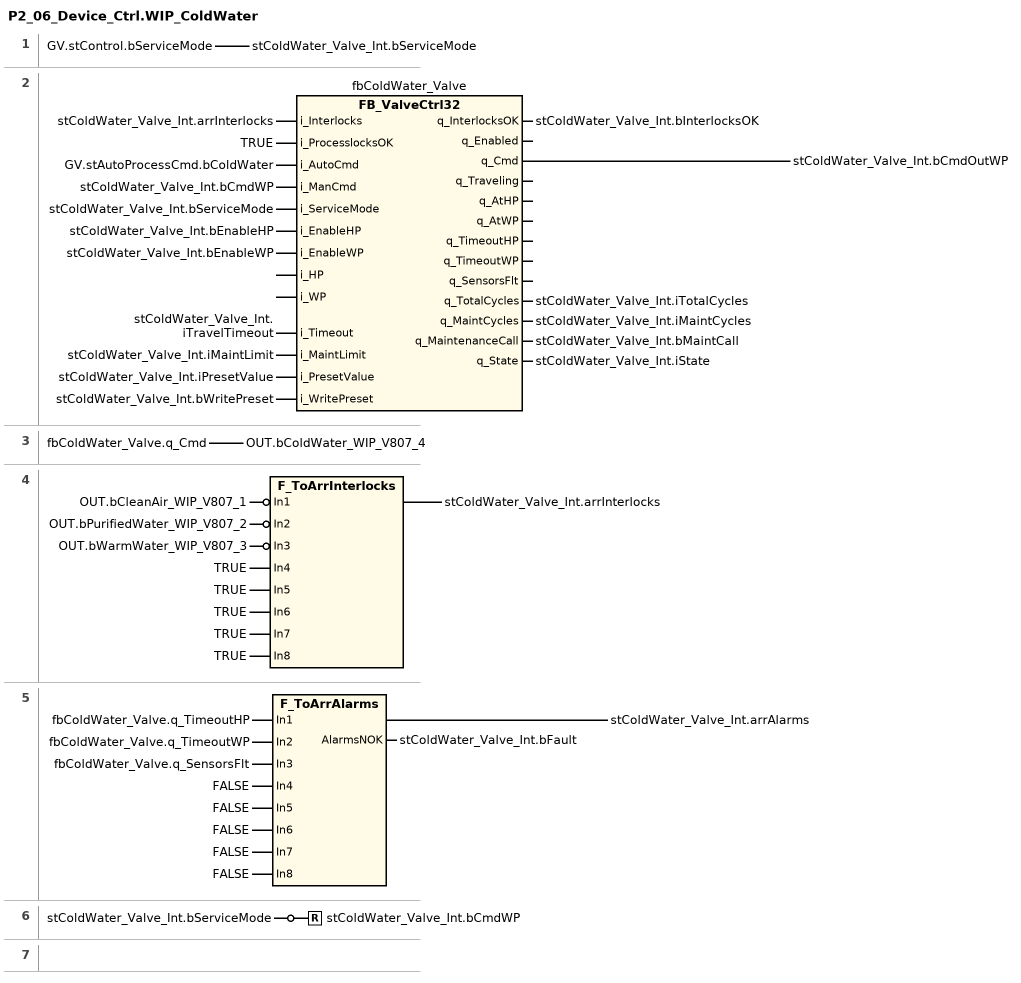
// NETWORK 1
stColdWater_Valve_Int.bServiceMode := GV.stControl.bServiceMode;

// NETWORK 2
fbColdWater_Valve(
    i_Interlocks := stColdWater_Valve_Int.arrInterlocks,
    i_ProcesslocksOK := TRUE,
    i_AutoCmd := GV.stAutoProcessCmd.bColdWater,
    i_ManCmd := stColdWater_Valve_Int.bCmdWP,
    i_ServiceMode := stColdWater_Valve_Int.bServiceMode,
    i_EnableHP := stColdWater_Valve_Int.bEnableHP,
    i_EnableWP := stColdWater_Valve_Int.bEnableWP,
    i_Timeout := stColdWater_Valve_Int.iTravelTimeout,
    i_MaintLimit := stColdWater_Valve_Int.iMaintLimit,
    i_PresetValue := stColdWater_Valve_Int.iPresetValue,
    i_WritePreset := stColdWater_Valve_Int.bWritePreset,
    q_InterlocksOK => stColdWater_Valve_Int.bInterlocksOK,
    q_TotalCycles => stColdWater_Valve_Int.iTotalCycles,
    q_MaintCycles => stColdWater_Valve_Int.iMaintCycles,
    q_MaintenanceCall => stColdWater_Valve_Int.bMaintCall,
    q_State => stColdWater_Valve_Int.iState); // FB_ValveCtrl32
stColdWater_Valve_Int.bCmdOutWP := fbColdWater_Valve.q_Cmd;

// NETWORK 3
OUT.bColdWater_WIP_V807_4 := fbColdWater_Valve.q_Cmd;

// NETWORK 4
stColdWater_Valve_Int.arrInterlocks := F_ToArrInterlocks(In1 := NOT OUT.bCleanAir_WIP_V807_1, In2 := NOT OUT.bPurifiedWater_WIP_V807_2, In3 := NOT OUT.bWarmWater_WIP_V807_3, In4 := TRUE, In5 := TRUE, In6 := TRUE, In7 := TRUE, In8 := TRUE);

// NETWORK 5
stColdWater_Valve_Int.arrAlarms := F_ToArrAlarms(In1 := fbColdWater_Valve.q_TimeoutHP, In2 := fbColdWater_Valve.q_TimeoutWP, In3 := fbColdWater_Valve.q_SensorsFlt, In4 := FALSE, In5 := FALSE, In6 := FALSE, In7 := FALSE, In8 := FALSE, AlarmsNOK => stColdWater_Valve_Int.bFault);

// NETWORK 6
stColdWater_Valve_Int.bCmdWP R= NOT stColdWater_Valve_Int.bServiceMode;

// NETWORK 7
END_ACTION

ACTION WIP_MainDrain:
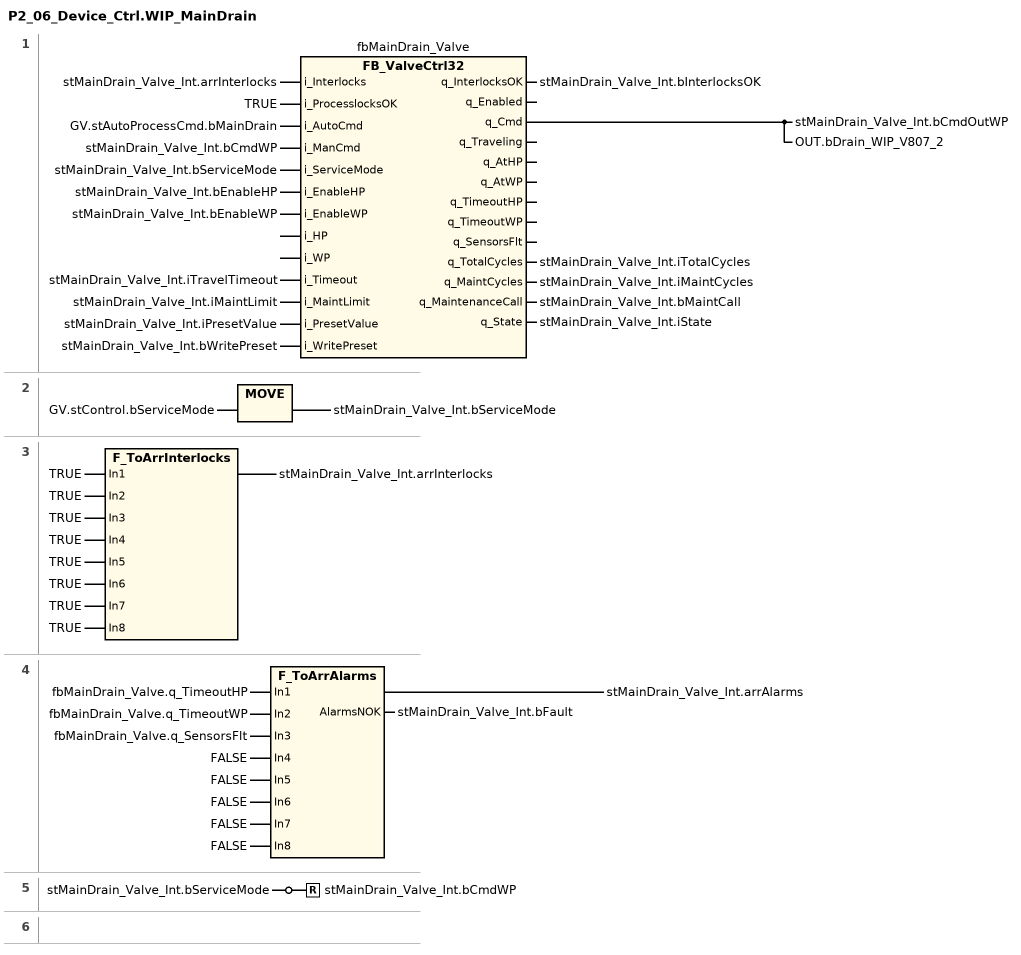
// NETWORK 1
fbMainDrain_Valve(
    i_Interlocks := stMainDrain_Valve_Int.arrInterlocks,
    i_ProcesslocksOK := TRUE,
    i_AutoCmd := GV.stAutoProcessCmd.bMainDrain,
    i_ManCmd := stMainDrain_Valve_Int.bCmdWP,
    i_ServiceMode := stMainDrain_Valve_Int.bServiceMode,
    i_EnableHP := stMainDrain_Valve_Int.bEnableHP,
    i_EnableWP := stMainDrain_Valve_Int.bEnableWP,
    i_Timeout := stMainDrain_Valve_Int.iTravelTimeout,
    i_MaintLimit := stMainDrain_Valve_Int.iMaintLimit,
    i_PresetValue := stMainDrain_Valve_Int.iPresetValue,
    i_WritePreset := stMainDrain_Valve_Int.bWritePreset,
    q_InterlocksOK => stMainDrain_Valve_Int.bInterlocksOK,
    q_TotalCycles => stMainDrain_Valve_Int.iTotalCycles,
    q_MaintCycles => stMainDrain_Valve_Int.iMaintCycles,
    q_MaintenanceCall => stMainDrain_Valve_Int.bMaintCall,
    q_State => stMainDrain_Valve_Int.iState); // FB_ValveCtrl32
stMainDrain_Valve_Int.bCmdOutWP := fbMainDrain_Valve.q_Cmd;
OUT.bDrain_WIP_V807_2 := fbMainDrain_Valve.q_Cmd;

// NETWORK 2
stMainDrain_Valve_Int.bServiceMode := GV.stControl.bServiceMode;

// NETWORK 3
stMainDrain_Valve_Int.arrInterlocks := F_ToArrInterlocks(In1 := TRUE, In2 := TRUE, In3 := TRUE, In4 := TRUE, In5 := TRUE, In6 := TRUE, In7 := TRUE, In8 := TRUE);

// NETWORK 4
stMainDrain_Valve_Int.arrAlarms := F_ToArrAlarms(In1 := fbMainDrain_Valve.q_TimeoutHP, In2 := fbMainDrain_Valve.q_TimeoutWP, In3 := fbMainDrain_Valve.q_SensorsFlt, In4 := FALSE, In5 := FALSE, In6 := FALSE, In7 := FALSE, In8 := FALSE, AlarmsNOK => stMainDrain_Valve_Int.bFault);

// NETWORK 5
stMainDrain_Valve_Int.bCmdWP R= NOT stMainDrain_Valve_Int.bServiceMode;

// NETWORK 6
END_ACTION

ACTION WIP_Mixer:
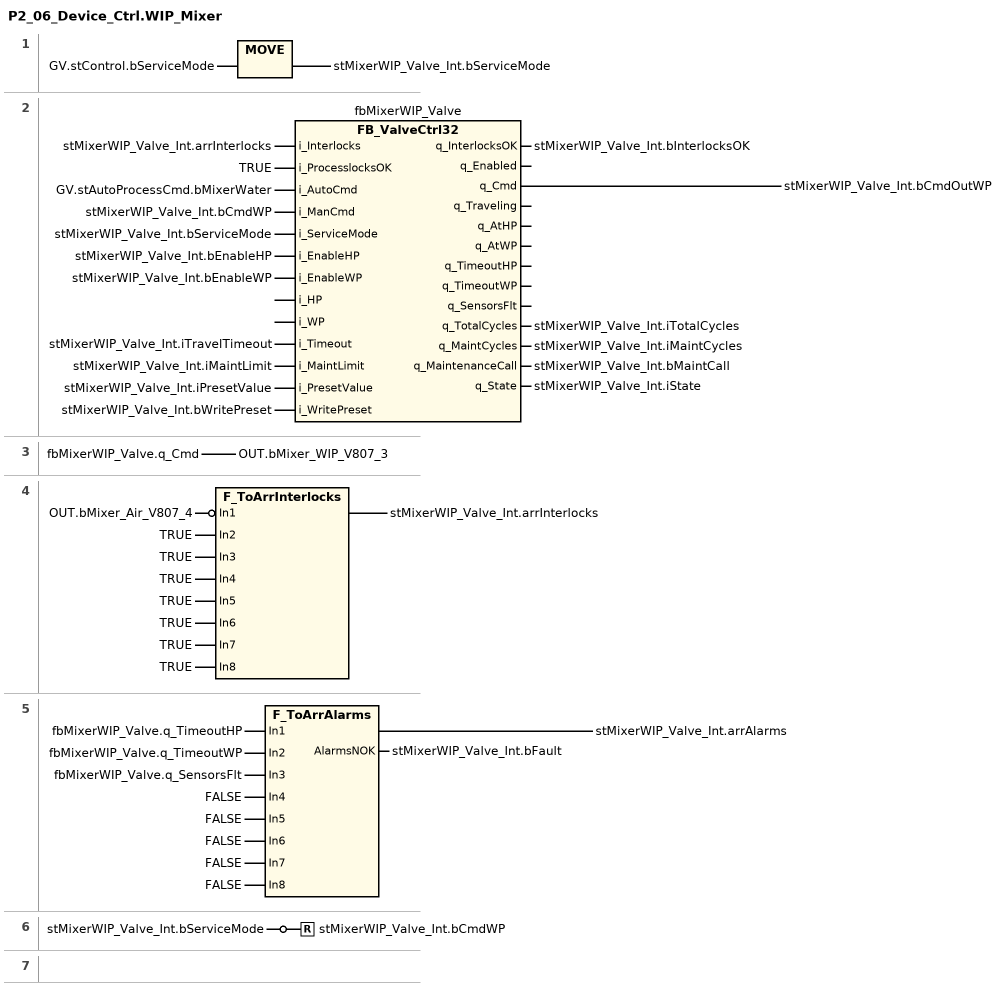
// NETWORK 1
stMixerWIP_Valve_Int.bServiceMode := GV.stControl.bServiceMode;

// NETWORK 2
fbMixerWIP_Valve(
    i_Interlocks := stMixerWIP_Valve_Int.arrInterlocks,
    i_ProcesslocksOK := TRUE,
    i_AutoCmd := GV.stAutoProcessCmd.bMixerWater,
    i_ManCmd := stMixerWIP_Valve_Int.bCmdWP,
    i_ServiceMode := stMixerWIP_Valve_Int.bServiceMode,
    i_EnableHP := stMixerWIP_Valve_Int.bEnableHP,
    i_EnableWP := stMixerWIP_Valve_Int.bEnableWP,
    i_Timeout := stMixerWIP_Valve_Int.iTravelTimeout,
    i_MaintLimit := stMixerWIP_Valve_Int.iMaintLimit,
    i_PresetValue := stMixerWIP_Valve_Int.iPresetValue,
    i_WritePreset := stMixerWIP_Valve_Int.bWritePreset,
    q_InterlocksOK => stMixerWIP_Valve_Int.bInterlocksOK,
    q_TotalCycles => stMixerWIP_Valve_Int.iTotalCycles,
    q_MaintCycles => stMixerWIP_Valve_Int.iMaintCycles,
    q_MaintenanceCall => stMixerWIP_Valve_Int.bMaintCall,
    q_State => stMixerWIP_Valve_Int.iState); // FB_ValveCtrl32
stMixerWIP_Valve_Int.bCmdOutWP := fbMixerWIP_Valve.q_Cmd;

// NETWORK 3
OUT.bMixer_WIP_V807_3 := fbMixerWIP_Valve.q_Cmd;

// NETWORK 4
stMixerWIP_Valve_Int.arrInterlocks := F_ToArrInterlocks(In1 := NOT OUT.bMixer_Air_V807_4, In2 := TRUE, In3 := TRUE, In4 := TRUE, In5 := TRUE, In6 := TRUE, In7 := TRUE, In8 := TRUE);

// NETWORK 5
stMixerWIP_Valve_Int.arrAlarms := F_ToArrAlarms(In1 := fbMixerWIP_Valve.q_TimeoutHP, In2 := fbMixerWIP_Valve.q_TimeoutWP, In3 := fbMixerWIP_Valve.q_SensorsFlt, In4 := FALSE, In5 := FALSE, In6 := FALSE, In7 := FALSE, In8 := FALSE, AlarmsNOK => stMixerWIP_Valve_Int.bFault);

// NETWORK 6
stMixerWIP_Valve_Int.bCmdWP R= NOT stMixerWIP_Valve_Int.bServiceMode;

// NETWORK 7
END_ACTION

ACTION WIP_PurifiedWater:
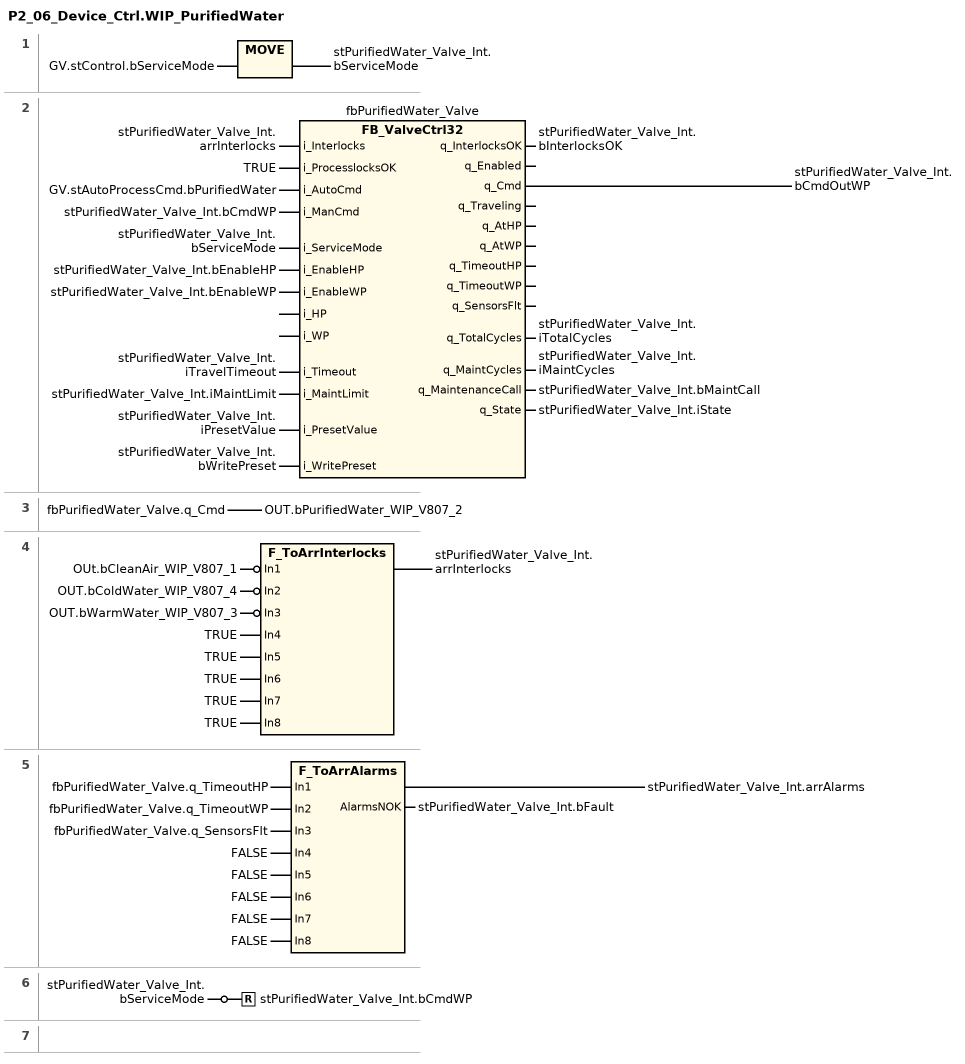
// NETWORK 1
stPurifiedWater_Valve_Int.bServiceMode := GV.stControl.bServiceMode;

// NETWORK 2
fbPurifiedWater_Valve(
    i_Interlocks := stPurifiedWater_Valve_Int.arrInterlocks,
    i_ProcesslocksOK := TRUE,
    i_AutoCmd := GV.stAutoProcessCmd.bPurifiedWater,
    i_ManCmd := stPurifiedWater_Valve_Int.bCmdWP,
    i_ServiceMode := stPurifiedWater_Valve_Int.bServiceMode,
    i_EnableHP := stPurifiedWater_Valve_Int.bEnableHP,
    i_EnableWP := stPurifiedWater_Valve_Int.bEnableWP,
    i_Timeout := stPurifiedWater_Valve_Int.iTravelTimeout,
    i_MaintLimit := stPurifiedWater_Valve_Int.iMaintLimit,
    i_PresetValue := stPurifiedWater_Valve_Int.iPresetValue,
    i_WritePreset := stPurifiedWater_Valve_Int.bWritePreset,
    q_InterlocksOK => stPurifiedWater_Valve_Int.bInterlocksOK,
    q_TotalCycles => stPurifiedWater_Valve_Int.iTotalCycles,
    q_MaintCycles => stPurifiedWater_Valve_Int.iMaintCycles,
    q_MaintenanceCall => stPurifiedWater_Valve_Int.bMaintCall,
    q_State => stPurifiedWater_Valve_Int.iState); // FB_ValveCtrl32
stPurifiedWater_Valve_Int.bCmdOutWP := fbPurifiedWater_Valve.q_Cmd;

// NETWORK 3
OUT.bPurifiedWater_WIP_V807_2 := fbPurifiedWater_Valve.q_Cmd;

// NETWORK 4
stPurifiedWater_Valve_Int.arrInterlocks := F_ToArrInterlocks(In1 := NOT OUt.bCleanAir_WIP_V807_1, In2 := NOT OUT.bColdWater_WIP_V807_4, In3 := NOT OUT.bWarmWater_WIP_V807_3, In4 := TRUE, In5 := TRUE, In6 := TRUE, In7 := TRUE, In8 := TRUE);

// NETWORK 5
stPurifiedWater_Valve_Int.arrAlarms := F_ToArrAlarms(In1 := fbPurifiedWater_Valve.q_TimeoutHP, In2 := fbPurifiedWater_Valve.q_TimeoutWP, In3 := fbPurifiedWater_Valve.q_SensorsFlt, In4 := FALSE, In5 := FALSE, In6 := FALSE, In7 := FALSE, In8 := FALSE, AlarmsNOK => stPurifiedWater_Valve_Int.bFault);

// NETWORK 6
stPurifiedWater_Valve_Int.bCmdWP R= NOT stPurifiedWater_Valve_Int.bServiceMode;

// NETWORK 7
END_ACTION

ACTION WIP_SP:
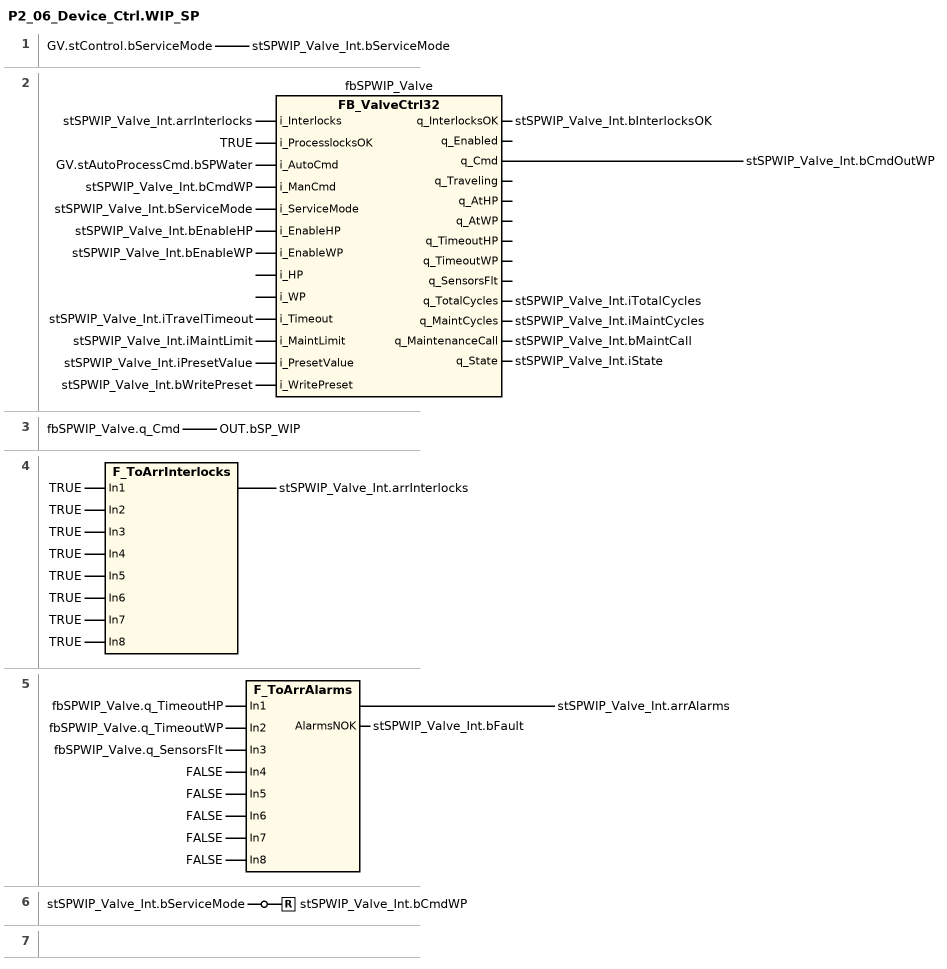
// NETWORK 1
stSPWIP_Valve_Int.bServiceMode := GV.stControl.bServiceMode;

// NETWORK 2
fbSPWIP_Valve(
    i_Interlocks := stSPWIP_Valve_Int.arrInterlocks,
    i_ProcesslocksOK := TRUE,
    i_AutoCmd := GV.stAutoProcessCmd.bSPWater,
    i_ManCmd := stSPWIP_Valve_Int.bCmdWP,
    i_ServiceMode := stSPWIP_Valve_Int.bServiceMode,
    i_EnableHP := stSPWIP_Valve_Int.bEnableHP,
    i_EnableWP := stSPWIP_Valve_Int.bEnableWP,
    i_Timeout := stSPWIP_Valve_Int.iTravelTimeout,
    i_MaintLimit := stSPWIP_Valve_Int.iMaintLimit,
    i_PresetValue := stSPWIP_Valve_Int.iPresetValue,
    i_WritePreset := stSPWIP_Valve_Int.bWritePreset,
    q_InterlocksOK => stSPWIP_Valve_Int.bInterlocksOK,
    q_TotalCycles => stSPWIP_Valve_Int.iTotalCycles,
    q_MaintCycles => stSPWIP_Valve_Int.iMaintCycles,
    q_MaintenanceCall => stSPWIP_Valve_Int.bMaintCall,
    q_State => stSPWIP_Valve_Int.iState); // FB_ValveCtrl32
stSPWIP_Valve_Int.bCmdOutWP := fbSPWIP_Valve.q_Cmd;

// NETWORK 3
OUT.bSP_WIP := fbSPWIP_Valve.q_Cmd;

// NETWORK 4
stSPWIP_Valve_Int.arrInterlocks := F_ToArrInterlocks(In1 := TRUE, In2 := TRUE, In3 := TRUE, In4 := TRUE, In5 := TRUE, In6 := TRUE, In7 := TRUE, In8 := TRUE);

// NETWORK 5
stSPWIP_Valve_Int.arrAlarms := F_ToArrAlarms(In1 := fbSPWIP_Valve.q_TimeoutHP, In2 := fbSPWIP_Valve.q_TimeoutWP, In3 := fbSPWIP_Valve.q_SensorsFlt, In4 := FALSE, In5 := FALSE, In6 := FALSE, In7 := FALSE, In8 := FALSE, AlarmsNOK => stSPWIP_Valve_Int.bFault);

// NETWORK 6
stSPWIP_Valve_Int.bCmdWP R= NOT stSPWIP_Valve_Int.bServiceMode;

// NETWORK 7
END_ACTION

ACTION WIP_SPDrain:
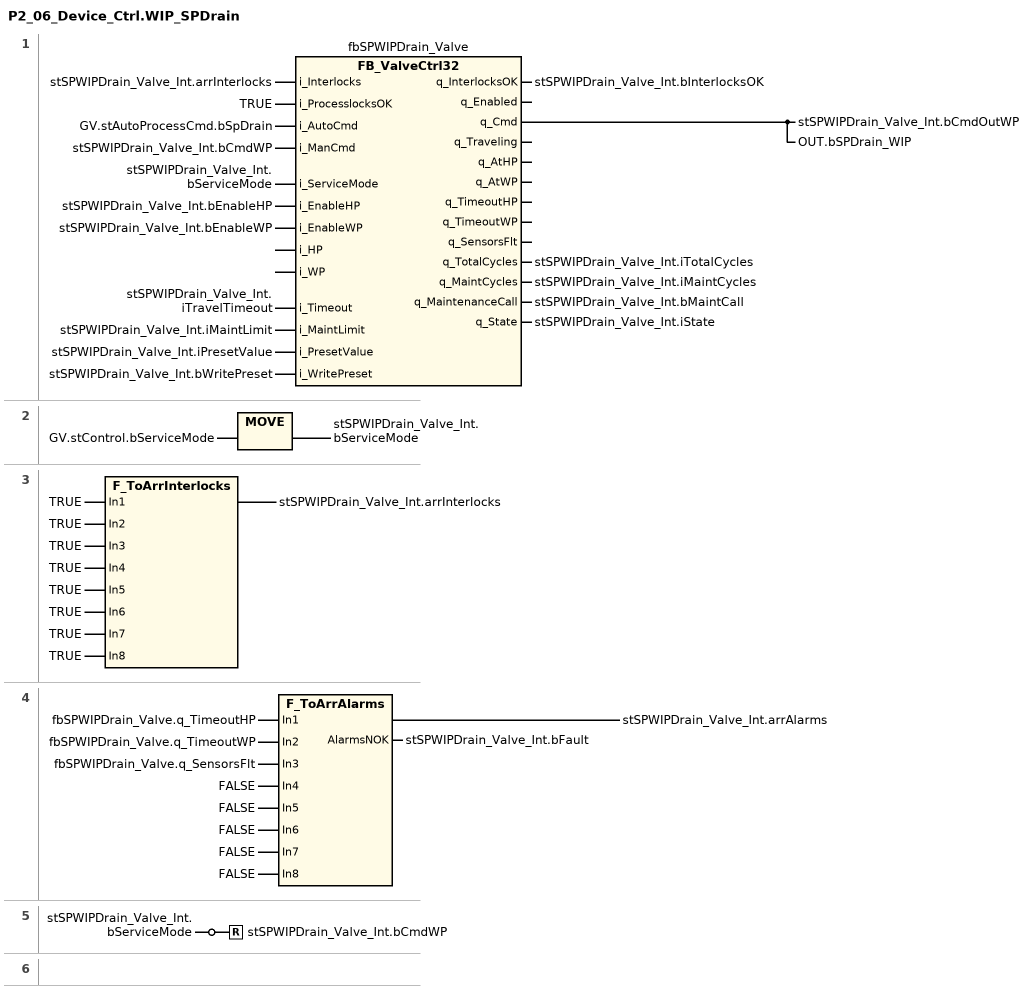
// NETWORK 1
fbSPWIPDrain_Valve(
    i_Interlocks := stSPWIPDrain_Valve_Int.arrInterlocks,
    i_ProcesslocksOK := TRUE,
    i_AutoCmd := GV.stAutoProcessCmd.bSpDrain,
    i_ManCmd := stSPWIPDrain_Valve_Int.bCmdWP,
    i_ServiceMode := stSPWIPDrain_Valve_Int.bServiceMode,
    i_EnableHP := stSPWIPDrain_Valve_Int.bEnableHP,
    i_EnableWP := stSPWIPDrain_Valve_Int.bEnableWP,
    i_Timeout := stSPWIPDrain_Valve_Int.iTravelTimeout,
    i_MaintLimit := stSPWIPDrain_Valve_Int.iMaintLimit,
    i_PresetValue := stSPWIPDrain_Valve_Int.iPresetValue,
    i_WritePreset := stSPWIPDrain_Valve_Int.bWritePreset,
    q_InterlocksOK => stSPWIPDrain_Valve_Int.bInterlocksOK,
    q_TotalCycles => stSPWIPDrain_Valve_Int.iTotalCycles,
    q_MaintCycles => stSPWIPDrain_Valve_Int.iMaintCycles,
    q_MaintenanceCall => stSPWIPDrain_Valve_Int.bMaintCall,
    q_State => stSPWIPDrain_Valve_Int.iState); // FB_ValveCtrl32
stSPWIPDrain_Valve_Int.bCmdOutWP := fbSPWIPDrain_Valve.q_Cmd;
OUT.bSPDrain_WIP := fbSPWIPDrain_Valve.q_Cmd;

// NETWORK 2
stSPWIPDrain_Valve_Int.bServiceMode := GV.stControl.bServiceMode;

// NETWORK 3
stSPWIPDrain_Valve_Int.arrInterlocks := F_ToArrInterlocks(In1 := TRUE, In2 := TRUE, In3 := TRUE, In4 := TRUE, In5 := TRUE, In6 := TRUE, In7 := TRUE, In8 := TRUE);

// NETWORK 4
stSPWIPDrain_Valve_Int.arrAlarms := F_ToArrAlarms(In1 := fbSPWIPDrain_Valve.q_TimeoutHP, In2 := fbSPWIPDrain_Valve.q_TimeoutWP, In3 := fbSPWIPDrain_Valve.q_SensorsFlt, In4 := FALSE, In5 := FALSE, In6 := FALSE, In7 := FALSE, In8 := FALSE, AlarmsNOK => stSPWIPDrain_Valve_Int.bFault);

// NETWORK 5
stSPWIPDrain_Valve_Int.bCmdWP R= NOT stSPWIPDrain_Valve_Int.bServiceMode;

// NETWORK 6
END_ACTION

ACTION WIP_WarmWater:
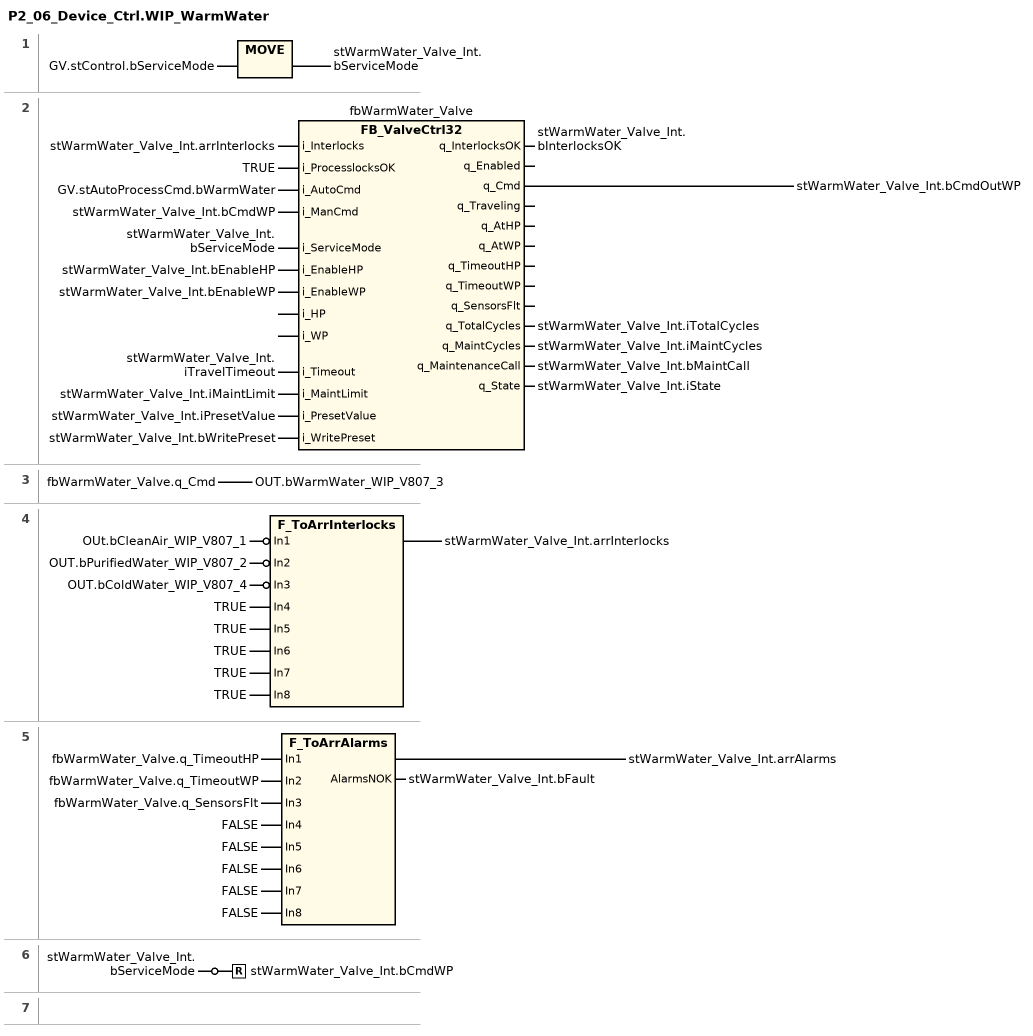
// NETWORK 1
stWarmWater_Valve_Int.bServiceMode := GV.stControl.bServiceMode;

// NETWORK 2
fbWarmWater_Valve(
    i_Interlocks := stWarmWater_Valve_Int.arrInterlocks,
    i_ProcesslocksOK := TRUE,
    i_AutoCmd := GV.stAutoProcessCmd.bWarmWater,
    i_ManCmd := stWarmWater_Valve_Int.bCmdWP,
    i_ServiceMode := stWarmWater_Valve_Int.bServiceMode,
    i_EnableHP := stWarmWater_Valve_Int.bEnableHP,
    i_EnableWP := stWarmWater_Valve_Int.bEnableWP,
    i_Timeout := stWarmWater_Valve_Int.iTravelTimeout,
    i_MaintLimit := stWarmWater_Valve_Int.iMaintLimit,
    i_PresetValue := stWarmWater_Valve_Int.iPresetValue,
    i_WritePreset := stWarmWater_Valve_Int.bWritePreset,
    q_InterlocksOK => stWarmWater_Valve_Int.bInterlocksOK,
    q_TotalCycles => stWarmWater_Valve_Int.iTotalCycles,
    q_MaintCycles => stWarmWater_Valve_Int.iMaintCycles,
    q_MaintenanceCall => stWarmWater_Valve_Int.bMaintCall,
    q_State => stWarmWater_Valve_Int.iState); // FB_ValveCtrl32
stWarmWater_Valve_Int.bCmdOutWP := fbWarmWater_Valve.q_Cmd;

// NETWORK 3
OUT.bWarmWater_WIP_V807_3 := fbWarmWater_Valve.q_Cmd;

// NETWORK 4
stWarmWater_Valve_Int.arrInterlocks := F_ToArrInterlocks(In1 := NOT OUt.bCleanAir_WIP_V807_1, In2 := NOT OUT.bPurifiedWater_WIP_V807_2, In3 := NOT OUT.bColdWater_WIP_V807_4, In4 := TRUE, In5 := TRUE, In6 := TRUE, In7 := TRUE, In8 := TRUE);

// NETWORK 5
stWarmWater_Valve_Int.arrAlarms := F_ToArrAlarms(In1 := fbWarmWater_Valve.q_TimeoutHP, In2 := fbWarmWater_Valve.q_TimeoutWP, In3 := fbWarmWater_Valve.q_SensorsFlt, In4 := FALSE, In5 := FALSE, In6 := FALSE, In7 := FALSE, In8 := FALSE, AlarmsNOK => stWarmWater_Valve_Int.bFault);

// NETWORK 6
stWarmWater_Valve_Int.bCmdWP R= NOT stWarmWater_Valve_Int.bServiceMode;

// NETWORK 7
END_ACTION

END_PROGRAM

(* stored: Version 1.1.0.1, ProductVersion 3.1.4024.12
   POU P2_06_Device_Ctrl: Id {b848229d-fdd9-4e19-9414-01f61c86ccbf}, SpecialFunc None
   Folder AOs: Id {608bfec8-bc32-444a-8134-3ab35aacd6a6}
   Folder Motors: Id {0f5cb510-5289-4d53-87e2-78ed15175d12}
   Folder PID: Id {2751b084-4cd1-492c-a53c-356d63484b9e}
   Folder Valves 3/2: Id {bb674119-6c88-40a3-be27-268a4dd9fd33}
   Folder Valves 5/2: Id {9b0d41c0-6d4e-4fd2-8824-076a74f2a694}
   Action Chopper: Id {2d8f816b-b933-4984-ad00-07e908d5d3de}
   Action Lid: Id {491d62ec-d387-457a-9976-34232c755ac7}
   Action Mixer: Id {3512aaa5-a8dc-4346-80c1-7e76533e4e9c}
   Action Outlet: Id {d32a22ed-4e27-4cd0-97c9-0ccceb757bc9}
   Action PROD_AirSeal: Id {7922e8d9-c076-455f-9922-77b247192270}
   Action PROD_Aspiration: Id {e75397af-9007-4695-a85b-8f6a160079b6}
   Action PROD_ChopperAir: Id {5d11882b-6017-4399-bce0-1efe374297c1}
   Action PROD_FilterClean: Id {19764443-8850-483e-b505-886b897a8290}
   Action PROD_MixerAir: Id {941f0b80-4bae-4a38-9907-d285663e9818}
   Action PROD_Vacuum: Id {5ffd15d5-28b0-4fe0-88df-882fe380b7f2}
   Action Pump: Id {bbb665a5-7aae-47f8-9ddb-4f318deec9df}
   Action Purge: Id {78b098b7-6c6c-4712-83ac-39d995aaa06e}
   Action Seal: Id {bafaecbb-1144-4caa-829c-1de45c85db08}
   Action Sieve: Id {0eebcfad-c23d-4bb0-bbd9-062fd6fe7971}
   Action SP_Mixer: Id {17d4f903-c2e0-468a-bb8e-34a92d815411}
   Action SP_Pressure: Id {5861b1c4-3b26-43c6-b7f1-8a9a674afb3d}
   Action SP_Temperature: Id {21c65aea-db54-42b1-98ee-1b2aa30e4430}
   Action Tool: Id {d59f3bae-2b32-4986-9d64-ad7b1e892dad}
   Action WIP_Chopper: Id {b699ca02-7d9b-4d3b-9c75-68dc0d67cdfb}
   Action WIP_CleaningAir: Id {72695808-e173-40ab-8997-8e505798f9bc}
   Action WIP_ColdWater: Id {7b31cd64-ac25-431e-8653-9ce5e57d21b0}
   Action WIP_MainDrain: Id {9d5e3aa8-3f2d-4cda-bab9-56656797783c}
   Action WIP_Mixer: Id {f73027eb-6238-4b96-9f5d-ff6ef5640f97}
   Action WIP_PurifiedWater: Id {b7c5df65-5e87-46d3-b86b-1bb5a7bb53b2}
   Action WIP_SP: Id {0f27f20a-3662-4793-a135-c04e943da321}
   Action WIP_SPDrain: Id {c2fb90c4-6c5a-4917-9e9d-e61c52ba9eca}
   Action WIP_WarmWater: Id {167d93e2-dc25-4548-b33f-620e2f9be2cb} *)
